//==================================================================================================
//								RJM Maszyny sp. z o.o.
//									04.06.2022
//	Sterowanie elektrozaworem  - 5 na 3 zapowietrzony 
//	nie ma podanych sygnałów na cewki powietrze jest podawane na siłownik (sterowanie odwrotne)
// 	v1.0	|| TC v 3.1.4024.22		|| - pierwsza wersja
//==================================================================================================
FUNCTION_BLOCK FB_Elektrozawor_5na3_Zapowietrzony IMPLEMENTS ITF_Elektozawor
VAR
	bCewkaA							AT %Q*	: BOOL;		//Cewka sterująca wyjściem 2 - 0 do MAX
	bCewkaB							AT %Q*	: BOOL;		//Cewka sterująca wyjściem 4 - MAX do 0
END_VAR

(*==================================================================================================
								RJM Maszyny sp. z o.o.
									04.06.2022
	Sterowanie cewkami elektrozaworu 
 	v1.0	|| TC v 3.1.4024.22		|| - pierwsza wersja
==================================================================================================*)
METHOD Steruj : BOOL
VAR_INPUT
	bKierunekWstrone0						: BOOL;
	bKierunekWStroneMax						: BOOL;
END_VAR
IF (bKierunekWStroneMax AND NOT bCewkaA) THEN
	bCewkaB									:= TRUE;
END_IF
IF  (bKierunekWstrone0 AND bCewkaA) THEN
	bCewkaB									:= FALSE;
END_IF

IF (bKierunekWstrone0 AND NOT bCewkaB) THEN
	bCewkaA									:= TRUE;
END_IF
IF  (bKierunekWStroneMax AND bCewkaB) THEN
	bCewkaA									:= FALSE;
END_IF
END_METHOD

END_FUNCTION_BLOCK

(* stored: Version 1.1.0.1, ProductVersion 3.1.4024.11
   POU FB_Elektrozawor_5na3_Zapowietrzony: Id {02092997-3d4c-4ecc-9017-0b8b59f3f30c}, SpecialFunc None
   Method Steruj: Id {37d5f088-fcf3-4d28-8853-628bf30ffe90} *)
